(* CoDeSys 2.3 export: GLOBAL_VARIABLES_MODBUS.EXP *)

(* Global variable list: Global_Variables_MODBUS *)
VAR_GLOBAL CONSTANT
	uiMaxCurrentDeviceSpace: UDINT := 99;
END_VAR
